(*
A broadcastable wrapper for a `REAL` value. 
*)
FUNCTION_BLOCK RealArg IMPLEMENTS I_RealArg
VAR
	_val			: REAL;
	_bMut			: BOOL := FALSE;
END_VAR

(*
Enables external modification of the internal value.
*)
METHOD AllowMut
_bMut := TRUE;
END_METHOD

(*
Disables external modification of the internal value.
*)
METHOD BlockMut
_bMut := FALSE;
END_METHOD

(*
Reads the internal value.
*)
PROPERTY Get : REAL
GET
Get := _val;
END_GET
END_PROPERTY

(*
Returns TRUE if the value is mutable.
*)
PROPERTY IsMut : BOOL
GET
IsMut := _bMut;
END_GET
END_PROPERTY

(*
Directly modifies the internal value, bypassing any mutability restrictions.
*)
METHOD OpSet : I_Arg
VAR_INPUT
	newVal		: REAL;
END_VAR
_val := newVal;
OpSet := THIS^;
END_METHOD

(*
Modifies the internal value.  
Returns:
- `Ok` - Upon successful modification.
- `Error` - If mutability is disabled.
*)
METHOD Set : Result
VAR_INPUT
	newVal		: REAL;
END_VAR
IF _bMut THEN
	_val := newVal;
	Set := Ok;
ELSE
	Set := Error;
END_IF
END_METHOD

END_FUNCTION_BLOCK

(* stored: Version 1.1.0.1
   POU RealArg: Id {38529bd9-c359-45c1-b5b2-c8912304cfc4}, SpecialFunc None
   Method AllowMut: Id {33cc2f5e-f55f-406c-b986-bda9e36cd320}
   Method BlockMut: Id {e3c89fa0-d5d9-42e4-b929-3ef4f5ef6131}
   Property Get: Id {ae04f6bf-9d46-4e43-8f76-e74798a0f7a4}
   Get Get: Id {9d27641c-cc29-401f-be07-96a0943c27c6}
   Property IsMut: Id {f5970024-1c3d-4917-8973-7bbd20b80745}
   Get Get: Id {71d859b1-dcc3-400c-876c-2f22313c376b}
   Method OpSet: Id {a019296d-a8e5-4ec4-9044-32d2ebfafdc0}
   Method Set: Id {a738a525-d9de-43b0-b302-91bcc30df04a} *)
